// TIA Portal V17 export
// export: Created 2024-09-02T12:50:12.8547271Z, ExportSetting WithDefaults, DisplayName Totally Integrated Automation Portal, DisplayVersion V17, DisplayName TIA Portal Openness, DisplayVersion V17, DisplayName TIA Portal Version Control Interface, DisplayVersion V17, DisplayName STEP 7 Professional, DisplayVersion V17, DisplayName STEP 7 Safety, DisplayVersion V17, DisplayName WinCC Professional, DisplayVersion V17
FUNCTION_BLOCK "AnwFB_Prozess_FG02_BEA3_OP70"   // FB503, LAD
TITLE = Processing dates 2 / Bearbeitungsdaten 2
{ S7_Optimized_Access := 'TRUE' }
AUTHOR : VAF
FAMILY : PROZESS
NAME : PROZESS
VERSION : 0.1
// stored: AutoNumber false, IsIECCheckEnabled false, IsRetainMemResEnabled false, MemoryReserve 100, SetENOAutomatically false, UDAEnableTagReadback false
   VAR
      Station { S7_SetPoint := 'True'} : "SysFB_ProzessDatenStation";
      Gruppe_0 { S7_SetPoint := 'True'} : "SysFB_ProzessDatenGruppe";
      Gruppe_1 { S7_SetPoint := 'True'} : "SysFB_ProzessDatenGruppe";
      Gruppe_2 { S7_SetPoint := 'True'} : "SysFB_ProzessDatenGruppe";
      Gruppe_3 { S7_SetPoint := 'True'} : "SysFB_ProzessDatenGruppe";
   END_VAR
   VAR_TEMP
      t_VKE0 : Bool;
      t_VKE1 : Bool;
      t_Reset : Bool;
      t_Release_Hand_OK : Bool;
      t_Release_Deselect : Bool;
      t_Release_Select : Bool;
      t_Release_NOK_Retry : Bool;
      t_Release_NOK_Reject : Bool;
      t_Reset_Hand_OK : Bool;
      t_Reset_Deselect : Bool;
      t_RetVal_SFC : Int;
   END_VAR
BEGIN

REGION Network 1 (SCL): Reload TAF No/indetyficator / TAF-Nr/Bezeichner umladen
   "AnwDB_ProcessData_FG02_OP70".PROZESS[3].Process.PROC_NR := 3;

   "AnwDB_ProcessData_FG02_OP70".PROZESS[3].Process.DES[1] := 'T';
   "AnwDB_ProcessData_FG02_OP70".PROZESS[3].Process.DES[2] := 'i';
   "AnwDB_ProcessData_FG02_OP70".PROZESS[3].Process.DES[3] := 'g';
   "AnwDB_ProcessData_FG02_OP70".PROZESS[3].Process.DES[4] := 'h';
   "AnwDB_ProcessData_FG02_OP70".PROZESS[3].Process.DES[5] := 't';
   "AnwDB_ProcessData_FG02_OP70".PROZESS[3].Process.DES[6] := 'e';
   "AnwDB_ProcessData_FG02_OP70".PROZESS[3].Process.DES[7] := 'n';
   "AnwDB_ProcessData_FG02_OP70".PROZESS[3].Process.DES[8] := 'i';
   "AnwDB_ProcessData_FG02_OP70".PROZESS[3].Process.DES[9] := 'n';
   "AnwDB_ProcessData_FG02_OP70".PROZESS[3].Process.DES[10] := 'g';
   "AnwDB_ProcessData_FG02_OP70".PROZESS[3].Process.DES[11] := ' ';
   "AnwDB_ProcessData_FG02_OP70".PROZESS[3].Process.DES[12] := ' ';
   "AnwDB_ProcessData_FG02_OP70".PROZESS[3].Process.DES[13] := ' ';
   "AnwDB_ProcessData_FG02_OP70".PROZESS[3].Process.DES[14] := ' ';
   "AnwDB_ProcessData_FG02_OP70".PROZESS[3].Process.DES[15] := ' ';
   "AnwDB_ProcessData_FG02_OP70".PROZESS[3].Process.DES[16] := ' ';
   "AnwDB_ProcessData_FG02_OP70".PROZESS[3].Process.DES[17] := ' ';
   "AnwDB_ProcessData_FG02_OP70".PROZESS[3].Process.DES[18] := ' ';
   "AnwDB_ProcessData_FG02_OP70".PROZESS[3].Process.DES[19] := ' ';
   "AnwDB_ProcessData_FG02_OP70".PROZESS[3].Process.DES[20] := ' ';
   "AnwDB_ProcessData_FG02_OP70".PROZESS[3].Process.DES[21] := ' ';
   "AnwDB_ProcessData_FG02_OP70".PROZESS[3].Process.DES[22] := ' ';
END_REGION

REGION Network 2: VKE0/1
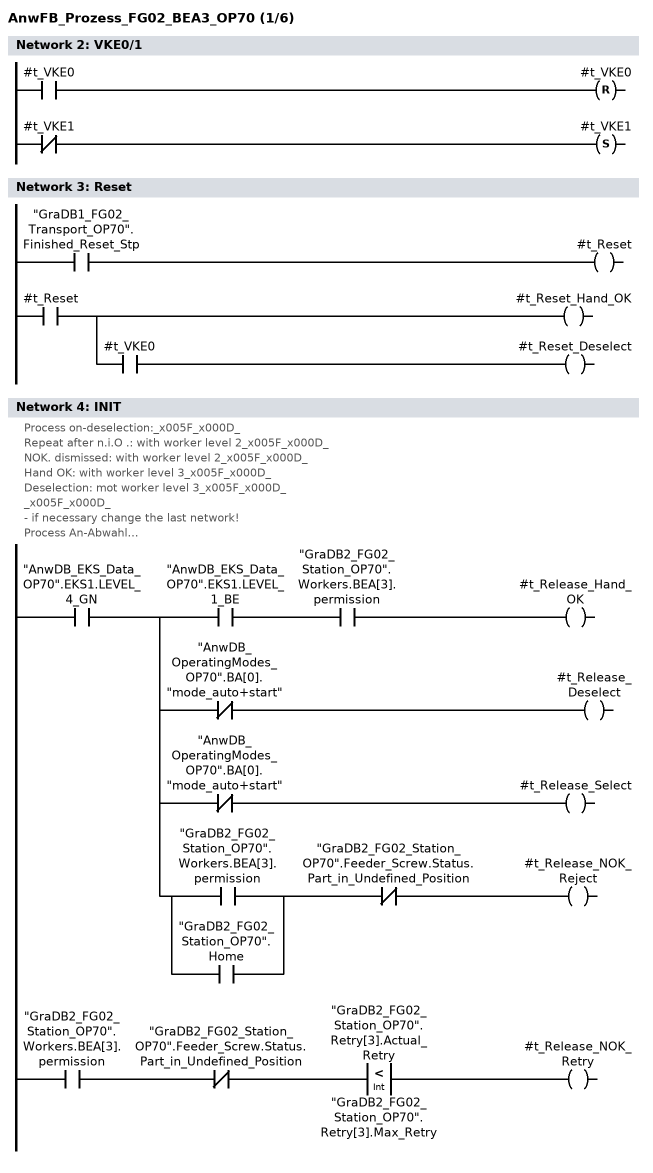
   RUNG wire#powerrail
      Contact( #t_VKE0 )
      R_Coil( #t_VKE0 )
   END_RUNG
   RUNG wire#powerrail
      I_Contact( #t_VKE1 )
      S_Coil( #t_VKE1 )
   END_RUNG
   // the same network as SCL:
   IF #t_VKE0 THEN #t_VKE0 := FALSE; END_IF;
   IF NOT #t_VKE1 THEN #t_VKE1 := TRUE; END_IF;
END_REGION

REGION Network 3: Reset
   RUNG wire#powerrail
      Contact( "GraDB1_FG02_Transport_OP70".Finished_Reset_Stp )
      Coil( #t_Reset )
   END_RUNG
   RUNG wire#powerrail
      Contact( #t_Reset )
      wire#w1
      Coil( #t_Reset_Hand_OK )
   END_RUNG
   RUNG wire#w1
      Contact( #t_VKE0 )
      Coil( #t_Reset_Deselect )
   END_RUNG
   // the same network as SCL:
   #t_Reset := "GraDB1_FG02_Transport_OP70".Finished_Reset_Stp;
   #t_Reset_Hand_OK := #t_Reset;
   #t_Reset_Deselect := #t_Reset AND #t_VKE0;
END_REGION

REGION Network 4: INIT
   // Process on-deselection:_x005F_x000D_
   // Repeat after n.i.O .: with worker level 2_x005F_x000D_
   // NOK. dismissed: with worker level 2_x005F_x000D_
   // Hand OK: with worker level 3_x005F_x000D_
   // Deselection: mot worker level 3_x005F_x000D_
   // _x005F_x000D_
   // - if necessary change the last network!
   // Process An-Abwahl:
   // Wiederholen nach n.i.O.: mit Werkerlevel 2
   // N.i.O. entlassen: mit Werkerlevel 2
   // Hand i.O: mit Werkerlevel 3
   // Abwahl: mot Werkerlevel 3
   // 
   // - bei Änderungen evtl.letztes Netzwerk anpassen !!
   RUNG wire#powerrail
      Contact( "AnwDB_EKS_Data_OP70".EKS1.LEVEL_4_GN )
      wire#w1
      Contact( "AnwDB_EKS_Data_OP70".EKS1.LEVEL_1_BE )
      Contact( "GraDB2_FG02_Station_OP70".Workers.BEA[3].permission )
      Coil( #t_Release_Hand_OK )
   END_RUNG
   RUNG wire#w1
      I_Contact( "AnwDB_OperatingModes_OP70".BA[0]."mode_auto+start" )
      Coil( #t_Release_Deselect )
   END_RUNG
   RUNG wire#w1
      I_Contact( "AnwDB_OperatingModes_OP70".BA[0]."mode_auto+start" )
      Coil( #t_Release_Select )
   END_RUNG
   RUNG wire#w1
      Contact( "GraDB2_FG02_Station_OP70".Workers.BEA[3].permission )
      wire#w2
      I_Contact( "GraDB2_FG02_Station_OP70".Feeder_Screw.Status.Part_in_Undefined_Position )
      Coil( #t_Release_NOK_Reject )
   END_RUNG
   RUNG wire#w1
      Contact( "GraDB2_FG02_Station_OP70".Home )
   END_RUNG wire#w2
   RUNG wire#powerrail
      Contact( "GraDB2_FG02_Station_OP70".Workers.BEA[3].permission )
      I_Contact( "GraDB2_FG02_Station_OP70".Feeder_Screw.Status.Part_in_Undefined_Position )
      { S7_Templates := "SrcType := Int" } LT_Contact(in1 := "GraDB2_FG02_Station_OP70".Retry[3].Actual_Retry, in2 := "GraDB2_FG02_Station_OP70".Retry[3].Max_Retry)
      Coil( #t_Release_NOK_Retry )
   END_RUNG
   // the same network as SCL:
   #t_Release_Hand_OK := "AnwDB_EKS_Data_OP70".EKS1.LEVEL_4_GN AND "AnwDB_EKS_Data_OP70".EKS1.LEVEL_1_BE AND "GraDB2_FG02_Station_OP70".Workers.BEA[3].permission;
   #t_Release_Deselect := "AnwDB_EKS_Data_OP70".EKS1.LEVEL_4_GN AND NOT "AnwDB_OperatingModes_OP70".BA[0]."mode_auto+start";
   #t_Release_Select := "AnwDB_EKS_Data_OP70".EKS1.LEVEL_4_GN AND NOT "AnwDB_OperatingModes_OP70".BA[0]."mode_auto+start";
   #t_Release_NOK_Reject := "AnwDB_EKS_Data_OP70".EKS1.LEVEL_4_GN AND ("GraDB2_FG02_Station_OP70".Workers.BEA[3].permission OR "GraDB2_FG02_Station_OP70".Home) AND NOT "GraDB2_FG02_Station_OP70".Feeder_Screw.Status.Part_in_Undefined_Position;
   #t_Release_NOK_Retry := "GraDB2_FG02_Station_OP70".Workers.BEA[3].permission AND NOT "GraDB2_FG02_Station_OP70".Feeder_Screw.Status.Part_in_Undefined_Position AND ("GraDB2_FG02_Station_OP70".Retry[3].Actual_Retry < "GraDB2_FG02_Station_OP70".Retry[3].Max_Retry);
END_REGION

REGION Network 5: Data Group 0 / Daten Gruppe 0
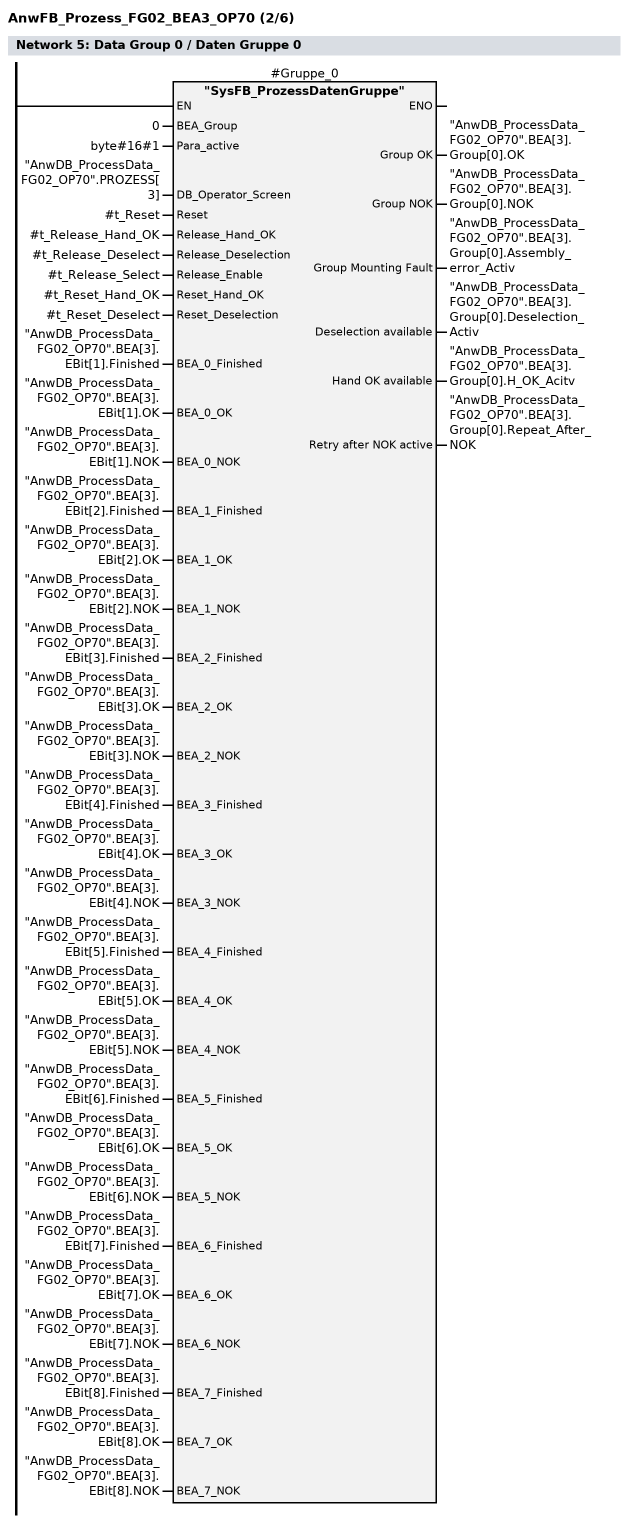
   RUNG wire#powerrail
      #Gruppe_0(BEA_Group := 0, Para_active := byte#16#1, DB_Operator_Screen := "AnwDB_ProcessData_FG02_OP70".PROZESS[3], Reset := #t_Reset, Release_Hand_OK := #t_Release_Hand_OK, Release_Deselection := #t_Release_Deselect, Release_Enable := #t_Release_Select, Reset_Hand_OK := #t_Reset_Hand_OK, Reset_Deselection := #t_Reset_Deselect, BEA_0_Finished := "AnwDB_ProcessData_FG02_OP70".BEA[3].EBit[1].Finished, BEA_0_OK := "AnwDB_ProcessData_FG02_OP70".BEA[3].EBit[1].OK, BEA_0_NOK := "AnwDB_ProcessData_FG02_OP70".BEA[3].EBit[1].NOK, BEA_1_Finished := "AnwDB_ProcessData_FG02_OP70".BEA[3].EBit[2].Finished, BEA_1_OK := "AnwDB_ProcessData_FG02_OP70".BEA[3].EBit[2].OK, BEA_1_NOK := "AnwDB_ProcessData_FG02_OP70".BEA[3].EBit[2].NOK, BEA_2_Finished := "AnwDB_ProcessData_FG02_OP70".BEA[3].EBit[3].Finished, BEA_2_OK := "AnwDB_ProcessData_FG02_OP70".BEA[3].EBit[3].OK, BEA_2_NOK := "AnwDB_ProcessData_FG02_OP70".BEA[3].EBit[3].NOK, BEA_3_Finished := "AnwDB_ProcessData_FG02_OP70".BEA[3].EBit[4].Finished, BEA_3_OK := "AnwDB_ProcessData_FG02_OP70".BEA[3].EBit[4].OK, BEA_3_NOK := "AnwDB_ProcessData_FG02_OP70".BEA[3].EBit[4].NOK, BEA_4_Finished := "AnwDB_ProcessData_FG02_OP70".BEA[3].EBit[5].Finished, BEA_4_OK := "AnwDB_ProcessData_FG02_OP70".BEA[3].EBit[5].OK, BEA_4_NOK := "AnwDB_ProcessData_FG02_OP70".BEA[3].EBit[5].NOK, BEA_5_Finished := "AnwDB_ProcessData_FG02_OP70".BEA[3].EBit[6].Finished, BEA_5_OK := "AnwDB_ProcessData_FG02_OP70".BEA[3].EBit[6].OK, BEA_5_NOK := "AnwDB_ProcessData_FG02_OP70".BEA[3].EBit[6].NOK, BEA_6_Finished := "AnwDB_ProcessData_FG02_OP70".BEA[3].EBit[7].Finished, BEA_6_OK := "AnwDB_ProcessData_FG02_OP70".BEA[3].EBit[7].OK, BEA_6_NOK := "AnwDB_ProcessData_FG02_OP70".BEA[3].EBit[7].NOK, BEA_7_Finished := "AnwDB_ProcessData_FG02_OP70".BEA[3].EBit[8].Finished, BEA_7_OK := "AnwDB_ProcessData_FG02_OP70".BEA[3].EBit[8].OK, BEA_7_NOK := "AnwDB_ProcessData_FG02_OP70".BEA[3].EBit[8].NOK, "Group OK" => "AnwDB_ProcessData_FG02_OP70".BEA[3].Group[0].OK, "Group NOK" => "AnwDB_ProcessData_FG02_OP70".BEA[3].Group[0].NOK, "Group Mounting Fault" => "AnwDB_ProcessData_FG02_OP70".BEA[3].Group[0].Assembly_error_Activ, "Deselection available" => "AnwDB_ProcessData_FG02_OP70".BEA[3].Group[0].Deselection_Activ, "Hand OK available" => "AnwDB_ProcessData_FG02_OP70".BEA[3].Group[0].H_OK_Acitv, "Retry after NOK active" => "AnwDB_ProcessData_FG02_OP70".BEA[3].Group[0].Repeat_After_NOK)
   END_RUNG
   // the same network as SCL:
   #Gruppe_0(BEA_Group := 0,   // "SysFB_ProzessDatenGruppe"
             Para_active := byte#16#1,
             DB_Operator_Screen := "AnwDB_ProcessData_FG02_OP70".PROZESS[3],
             Reset := #t_Reset,
             Release_Hand_OK := #t_Release_Hand_OK,
             Release_Deselection := #t_Release_Deselect,
             Release_Enable := #t_Release_Select,
             Reset_Hand_OK := #t_Reset_Hand_OK,
             Reset_Deselection := #t_Reset_Deselect,
             BEA_0_Finished := "AnwDB_ProcessData_FG02_OP70".BEA[3].EBit[1].Finished,
             BEA_0_OK := "AnwDB_ProcessData_FG02_OP70".BEA[3].EBit[1].OK,
             BEA_0_NOK := "AnwDB_ProcessData_FG02_OP70".BEA[3].EBit[1].NOK,
             BEA_1_Finished := "AnwDB_ProcessData_FG02_OP70".BEA[3].EBit[2].Finished,
             BEA_1_OK := "AnwDB_ProcessData_FG02_OP70".BEA[3].EBit[2].OK,
             BEA_1_NOK := "AnwDB_ProcessData_FG02_OP70".BEA[3].EBit[2].NOK,
             BEA_2_Finished := "AnwDB_ProcessData_FG02_OP70".BEA[3].EBit[3].Finished,
             BEA_2_OK := "AnwDB_ProcessData_FG02_OP70".BEA[3].EBit[3].OK,
             BEA_2_NOK := "AnwDB_ProcessData_FG02_OP70".BEA[3].EBit[3].NOK,
             BEA_3_Finished := "AnwDB_ProcessData_FG02_OP70".BEA[3].EBit[4].Finished,
             BEA_3_OK := "AnwDB_ProcessData_FG02_OP70".BEA[3].EBit[4].OK,
             BEA_3_NOK := "AnwDB_ProcessData_FG02_OP70".BEA[3].EBit[4].NOK,
             BEA_4_Finished := "AnwDB_ProcessData_FG02_OP70".BEA[3].EBit[5].Finished,
             BEA_4_OK := "AnwDB_ProcessData_FG02_OP70".BEA[3].EBit[5].OK,
             BEA_4_NOK := "AnwDB_ProcessData_FG02_OP70".BEA[3].EBit[5].NOK,
             BEA_5_Finished := "AnwDB_ProcessData_FG02_OP70".BEA[3].EBit[6].Finished,
             BEA_5_OK := "AnwDB_ProcessData_FG02_OP70".BEA[3].EBit[6].OK,
             BEA_5_NOK := "AnwDB_ProcessData_FG02_OP70".BEA[3].EBit[6].NOK,
             BEA_6_Finished := "AnwDB_ProcessData_FG02_OP70".BEA[3].EBit[7].Finished,
             BEA_6_OK := "AnwDB_ProcessData_FG02_OP70".BEA[3].EBit[7].OK,
             BEA_6_NOK := "AnwDB_ProcessData_FG02_OP70".BEA[3].EBit[7].NOK,
             BEA_7_Finished := "AnwDB_ProcessData_FG02_OP70".BEA[3].EBit[8].Finished,
             BEA_7_OK := "AnwDB_ProcessData_FG02_OP70".BEA[3].EBit[8].OK,
             BEA_7_NOK := "AnwDB_ProcessData_FG02_OP70".BEA[3].EBit[8].NOK,
             "Group OK" => "AnwDB_ProcessData_FG02_OP70".BEA[3].Group[0].OK,
             "Group NOK" => "AnwDB_ProcessData_FG02_OP70".BEA[3].Group[0].NOK,
             "Group Mounting Fault" => "AnwDB_ProcessData_FG02_OP70".BEA[3].Group[0].Assembly_error_Activ,
             "Deselection available" => "AnwDB_ProcessData_FG02_OP70".BEA[3].Group[0].Deselection_Activ,
             "Hand OK available" => "AnwDB_ProcessData_FG02_OP70".BEA[3].Group[0].H_OK_Acitv,
             "Retry after NOK active" => "AnwDB_ProcessData_FG02_OP70".BEA[3].Group[0].Repeat_After_NOK);
END_REGION

REGION Network 6: Data Group 1 / Daten Gruppe 1
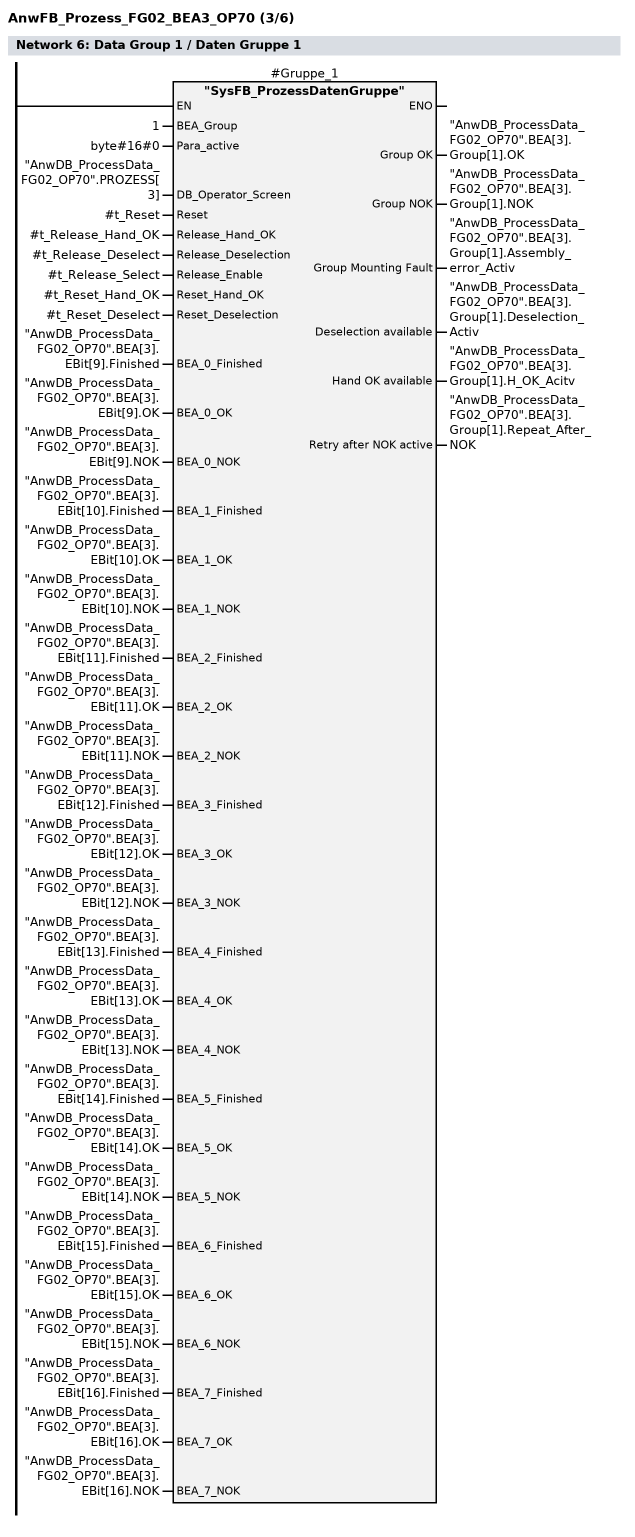
   RUNG wire#powerrail
      #Gruppe_1(BEA_Group := 1, Para_active := byte#16#0, DB_Operator_Screen := "AnwDB_ProcessData_FG02_OP70".PROZESS[3], Reset := #t_Reset, Release_Hand_OK := #t_Release_Hand_OK, Release_Deselection := #t_Release_Deselect, Release_Enable := #t_Release_Select, Reset_Hand_OK := #t_Reset_Hand_OK, Reset_Deselection := #t_Reset_Deselect, BEA_0_Finished := "AnwDB_ProcessData_FG02_OP70".BEA[3].EBit[9].Finished, BEA_0_OK := "AnwDB_ProcessData_FG02_OP70".BEA[3].EBit[9].OK, BEA_0_NOK := "AnwDB_ProcessData_FG02_OP70".BEA[3].EBit[9].NOK, BEA_1_Finished := "AnwDB_ProcessData_FG02_OP70".BEA[3].EBit[10].Finished, BEA_1_OK := "AnwDB_ProcessData_FG02_OP70".BEA[3].EBit[10].OK, BEA_1_NOK := "AnwDB_ProcessData_FG02_OP70".BEA[3].EBit[10].NOK, BEA_2_Finished := "AnwDB_ProcessData_FG02_OP70".BEA[3].EBit[11].Finished, BEA_2_OK := "AnwDB_ProcessData_FG02_OP70".BEA[3].EBit[11].OK, BEA_2_NOK := "AnwDB_ProcessData_FG02_OP70".BEA[3].EBit[11].NOK, BEA_3_Finished := "AnwDB_ProcessData_FG02_OP70".BEA[3].EBit[12].Finished, BEA_3_OK := "AnwDB_ProcessData_FG02_OP70".BEA[3].EBit[12].OK, BEA_3_NOK := "AnwDB_ProcessData_FG02_OP70".BEA[3].EBit[12].NOK, BEA_4_Finished := "AnwDB_ProcessData_FG02_OP70".BEA[3].EBit[13].Finished, BEA_4_OK := "AnwDB_ProcessData_FG02_OP70".BEA[3].EBit[13].OK, BEA_4_NOK := "AnwDB_ProcessData_FG02_OP70".BEA[3].EBit[13].NOK, BEA_5_Finished := "AnwDB_ProcessData_FG02_OP70".BEA[3].EBit[14].Finished, BEA_5_OK := "AnwDB_ProcessData_FG02_OP70".BEA[3].EBit[14].OK, BEA_5_NOK := "AnwDB_ProcessData_FG02_OP70".BEA[3].EBit[14].NOK, BEA_6_Finished := "AnwDB_ProcessData_FG02_OP70".BEA[3].EBit[15].Finished, BEA_6_OK := "AnwDB_ProcessData_FG02_OP70".BEA[3].EBit[15].OK, BEA_6_NOK := "AnwDB_ProcessData_FG02_OP70".BEA[3].EBit[15].NOK, BEA_7_Finished := "AnwDB_ProcessData_FG02_OP70".BEA[3].EBit[16].Finished, BEA_7_OK := "AnwDB_ProcessData_FG02_OP70".BEA[3].EBit[16].OK, BEA_7_NOK := "AnwDB_ProcessData_FG02_OP70".BEA[3].EBit[16].NOK, "Group OK" => "AnwDB_ProcessData_FG02_OP70".BEA[3].Group[1].OK, "Group NOK" => "AnwDB_ProcessData_FG02_OP70".BEA[3].Group[1].NOK, "Group Mounting Fault" => "AnwDB_ProcessData_FG02_OP70".BEA[3].Group[1].Assembly_error_Activ, "Deselection available" => "AnwDB_ProcessData_FG02_OP70".BEA[3].Group[1].Deselection_Activ, "Hand OK available" => "AnwDB_ProcessData_FG02_OP70".BEA[3].Group[1].H_OK_Acitv, "Retry after NOK active" => "AnwDB_ProcessData_FG02_OP70".BEA[3].Group[1].Repeat_After_NOK)
   END_RUNG
   // the same network as SCL:
   #Gruppe_1(BEA_Group := 1,   // "SysFB_ProzessDatenGruppe"
             Para_active := byte#16#0,
             DB_Operator_Screen := "AnwDB_ProcessData_FG02_OP70".PROZESS[3],
             Reset := #t_Reset,
             Release_Hand_OK := #t_Release_Hand_OK,
             Release_Deselection := #t_Release_Deselect,
             Release_Enable := #t_Release_Select,
             Reset_Hand_OK := #t_Reset_Hand_OK,
             Reset_Deselection := #t_Reset_Deselect,
             BEA_0_Finished := "AnwDB_ProcessData_FG02_OP70".BEA[3].EBit[9].Finished,
             BEA_0_OK := "AnwDB_ProcessData_FG02_OP70".BEA[3].EBit[9].OK,
             BEA_0_NOK := "AnwDB_ProcessData_FG02_OP70".BEA[3].EBit[9].NOK,
             BEA_1_Finished := "AnwDB_ProcessData_FG02_OP70".BEA[3].EBit[10].Finished,
             BEA_1_OK := "AnwDB_ProcessData_FG02_OP70".BEA[3].EBit[10].OK,
             BEA_1_NOK := "AnwDB_ProcessData_FG02_OP70".BEA[3].EBit[10].NOK,
             BEA_2_Finished := "AnwDB_ProcessData_FG02_OP70".BEA[3].EBit[11].Finished,
             BEA_2_OK := "AnwDB_ProcessData_FG02_OP70".BEA[3].EBit[11].OK,
             BEA_2_NOK := "AnwDB_ProcessData_FG02_OP70".BEA[3].EBit[11].NOK,
             BEA_3_Finished := "AnwDB_ProcessData_FG02_OP70".BEA[3].EBit[12].Finished,
             BEA_3_OK := "AnwDB_ProcessData_FG02_OP70".BEA[3].EBit[12].OK,
             BEA_3_NOK := "AnwDB_ProcessData_FG02_OP70".BEA[3].EBit[12].NOK,
             BEA_4_Finished := "AnwDB_ProcessData_FG02_OP70".BEA[3].EBit[13].Finished,
             BEA_4_OK := "AnwDB_ProcessData_FG02_OP70".BEA[3].EBit[13].OK,
             BEA_4_NOK := "AnwDB_ProcessData_FG02_OP70".BEA[3].EBit[13].NOK,
             BEA_5_Finished := "AnwDB_ProcessData_FG02_OP70".BEA[3].EBit[14].Finished,
             BEA_5_OK := "AnwDB_ProcessData_FG02_OP70".BEA[3].EBit[14].OK,
             BEA_5_NOK := "AnwDB_ProcessData_FG02_OP70".BEA[3].EBit[14].NOK,
             BEA_6_Finished := "AnwDB_ProcessData_FG02_OP70".BEA[3].EBit[15].Finished,
             BEA_6_OK := "AnwDB_ProcessData_FG02_OP70".BEA[3].EBit[15].OK,
             BEA_6_NOK := "AnwDB_ProcessData_FG02_OP70".BEA[3].EBit[15].NOK,
             BEA_7_Finished := "AnwDB_ProcessData_FG02_OP70".BEA[3].EBit[16].Finished,
             BEA_7_OK := "AnwDB_ProcessData_FG02_OP70".BEA[3].EBit[16].OK,
             BEA_7_NOK := "AnwDB_ProcessData_FG02_OP70".BEA[3].EBit[16].NOK,
             "Group OK" => "AnwDB_ProcessData_FG02_OP70".BEA[3].Group[1].OK,
             "Group NOK" => "AnwDB_ProcessData_FG02_OP70".BEA[3].Group[1].NOK,
             "Group Mounting Fault" => "AnwDB_ProcessData_FG02_OP70".BEA[3].Group[1].Assembly_error_Activ,
             "Deselection available" => "AnwDB_ProcessData_FG02_OP70".BEA[3].Group[1].Deselection_Activ,
             "Hand OK available" => "AnwDB_ProcessData_FG02_OP70".BEA[3].Group[1].H_OK_Acitv,
             "Retry after NOK active" => "AnwDB_ProcessData_FG02_OP70".BEA[3].Group[1].Repeat_After_NOK);
END_REGION

REGION Network 7: Data Group 2 / Daten Gruppe 2
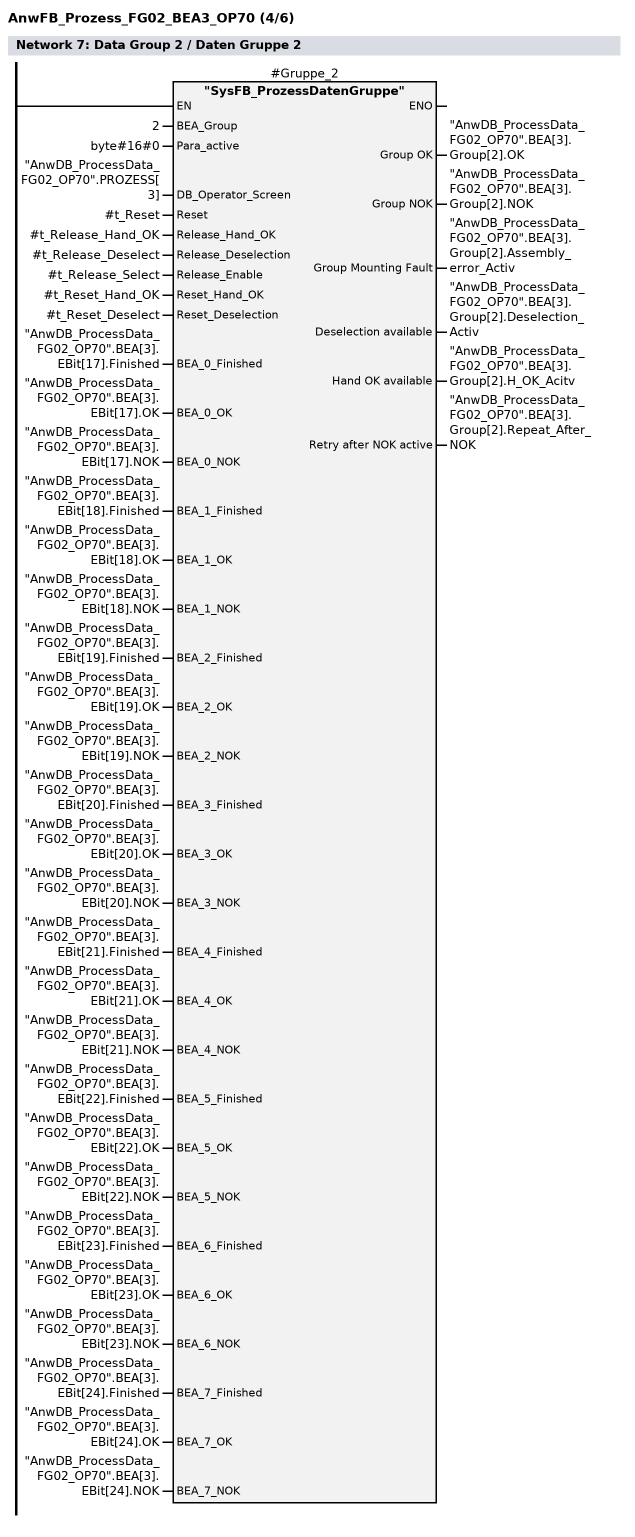
   RUNG wire#powerrail
      #Gruppe_2(BEA_Group := 2, Para_active := byte#16#0, DB_Operator_Screen := "AnwDB_ProcessData_FG02_OP70".PROZESS[3], Reset := #t_Reset, Release_Hand_OK := #t_Release_Hand_OK, Release_Deselection := #t_Release_Deselect, Release_Enable := #t_Release_Select, Reset_Hand_OK := #t_Reset_Hand_OK, Reset_Deselection := #t_Reset_Deselect, BEA_0_Finished := "AnwDB_ProcessData_FG02_OP70".BEA[3].EBit[17].Finished, BEA_0_OK := "AnwDB_ProcessData_FG02_OP70".BEA[3].EBit[17].OK, BEA_0_NOK := "AnwDB_ProcessData_FG02_OP70".BEA[3].EBit[17].NOK, BEA_1_Finished := "AnwDB_ProcessData_FG02_OP70".BEA[3].EBit[18].Finished, BEA_1_OK := "AnwDB_ProcessData_FG02_OP70".BEA[3].EBit[18].OK, BEA_1_NOK := "AnwDB_ProcessData_FG02_OP70".BEA[3].EBit[18].NOK, BEA_2_Finished := "AnwDB_ProcessData_FG02_OP70".BEA[3].EBit[19].Finished, BEA_2_OK := "AnwDB_ProcessData_FG02_OP70".BEA[3].EBit[19].OK, BEA_2_NOK := "AnwDB_ProcessData_FG02_OP70".BEA[3].EBit[19].NOK, BEA_3_Finished := "AnwDB_ProcessData_FG02_OP70".BEA[3].EBit[20].Finished, BEA_3_OK := "AnwDB_ProcessData_FG02_OP70".BEA[3].EBit[20].OK, BEA_3_NOK := "AnwDB_ProcessData_FG02_OP70".BEA[3].EBit[20].NOK, BEA_4_Finished := "AnwDB_ProcessData_FG02_OP70".BEA[3].EBit[21].Finished, BEA_4_OK := "AnwDB_ProcessData_FG02_OP70".BEA[3].EBit[21].OK, BEA_4_NOK := "AnwDB_ProcessData_FG02_OP70".BEA[3].EBit[21].NOK, BEA_5_Finished := "AnwDB_ProcessData_FG02_OP70".BEA[3].EBit[22].Finished, BEA_5_OK := "AnwDB_ProcessData_FG02_OP70".BEA[3].EBit[22].OK, BEA_5_NOK := "AnwDB_ProcessData_FG02_OP70".BEA[3].EBit[22].NOK, BEA_6_Finished := "AnwDB_ProcessData_FG02_OP70".BEA[3].EBit[23].Finished, BEA_6_OK := "AnwDB_ProcessData_FG02_OP70".BEA[3].EBit[23].OK, BEA_6_NOK := "AnwDB_ProcessData_FG02_OP70".BEA[3].EBit[23].NOK, BEA_7_Finished := "AnwDB_ProcessData_FG02_OP70".BEA[3].EBit[24].Finished, BEA_7_OK := "AnwDB_ProcessData_FG02_OP70".BEA[3].EBit[24].OK, BEA_7_NOK := "AnwDB_ProcessData_FG02_OP70".BEA[3].EBit[24].NOK, "Group OK" => "AnwDB_ProcessData_FG02_OP70".BEA[3].Group[2].OK, "Group NOK" => "AnwDB_ProcessData_FG02_OP70".BEA[3].Group[2].NOK, "Group Mounting Fault" => "AnwDB_ProcessData_FG02_OP70".BEA[3].Group[2].Assembly_error_Activ, "Deselection available" => "AnwDB_ProcessData_FG02_OP70".BEA[3].Group[2].Deselection_Activ, "Hand OK available" => "AnwDB_ProcessData_FG02_OP70".BEA[3].Group[2].H_OK_Acitv, "Retry after NOK active" => "AnwDB_ProcessData_FG02_OP70".BEA[3].Group[2].Repeat_After_NOK)
   END_RUNG
   // the same network as SCL:
   #Gruppe_2(BEA_Group := 2,   // "SysFB_ProzessDatenGruppe"
             Para_active := byte#16#0,
             DB_Operator_Screen := "AnwDB_ProcessData_FG02_OP70".PROZESS[3],
             Reset := #t_Reset,
             Release_Hand_OK := #t_Release_Hand_OK,
             Release_Deselection := #t_Release_Deselect,
             Release_Enable := #t_Release_Select,
             Reset_Hand_OK := #t_Reset_Hand_OK,
             Reset_Deselection := #t_Reset_Deselect,
             BEA_0_Finished := "AnwDB_ProcessData_FG02_OP70".BEA[3].EBit[17].Finished,
             BEA_0_OK := "AnwDB_ProcessData_FG02_OP70".BEA[3].EBit[17].OK,
             BEA_0_NOK := "AnwDB_ProcessData_FG02_OP70".BEA[3].EBit[17].NOK,
             BEA_1_Finished := "AnwDB_ProcessData_FG02_OP70".BEA[3].EBit[18].Finished,
             BEA_1_OK := "AnwDB_ProcessData_FG02_OP70".BEA[3].EBit[18].OK,
             BEA_1_NOK := "AnwDB_ProcessData_FG02_OP70".BEA[3].EBit[18].NOK,
             BEA_2_Finished := "AnwDB_ProcessData_FG02_OP70".BEA[3].EBit[19].Finished,
             BEA_2_OK := "AnwDB_ProcessData_FG02_OP70".BEA[3].EBit[19].OK,
             BEA_2_NOK := "AnwDB_ProcessData_FG02_OP70".BEA[3].EBit[19].NOK,
             BEA_3_Finished := "AnwDB_ProcessData_FG02_OP70".BEA[3].EBit[20].Finished,
             BEA_3_OK := "AnwDB_ProcessData_FG02_OP70".BEA[3].EBit[20].OK,
             BEA_3_NOK := "AnwDB_ProcessData_FG02_OP70".BEA[3].EBit[20].NOK,
             BEA_4_Finished := "AnwDB_ProcessData_FG02_OP70".BEA[3].EBit[21].Finished,
             BEA_4_OK := "AnwDB_ProcessData_FG02_OP70".BEA[3].EBit[21].OK,
             BEA_4_NOK := "AnwDB_ProcessData_FG02_OP70".BEA[3].EBit[21].NOK,
             BEA_5_Finished := "AnwDB_ProcessData_FG02_OP70".BEA[3].EBit[22].Finished,
             BEA_5_OK := "AnwDB_ProcessData_FG02_OP70".BEA[3].EBit[22].OK,
             BEA_5_NOK := "AnwDB_ProcessData_FG02_OP70".BEA[3].EBit[22].NOK,
             BEA_6_Finished := "AnwDB_ProcessData_FG02_OP70".BEA[3].EBit[23].Finished,
             BEA_6_OK := "AnwDB_ProcessData_FG02_OP70".BEA[3].EBit[23].OK,
             BEA_6_NOK := "AnwDB_ProcessData_FG02_OP70".BEA[3].EBit[23].NOK,
             BEA_7_Finished := "AnwDB_ProcessData_FG02_OP70".BEA[3].EBit[24].Finished,
             BEA_7_OK := "AnwDB_ProcessData_FG02_OP70".BEA[3].EBit[24].OK,
             BEA_7_NOK := "AnwDB_ProcessData_FG02_OP70".BEA[3].EBit[24].NOK,
             "Group OK" => "AnwDB_ProcessData_FG02_OP70".BEA[3].Group[2].OK,
             "Group NOK" => "AnwDB_ProcessData_FG02_OP70".BEA[3].Group[2].NOK,
             "Group Mounting Fault" => "AnwDB_ProcessData_FG02_OP70".BEA[3].Group[2].Assembly_error_Activ,
             "Deselection available" => "AnwDB_ProcessData_FG02_OP70".BEA[3].Group[2].Deselection_Activ,
             "Hand OK available" => "AnwDB_ProcessData_FG02_OP70".BEA[3].Group[2].H_OK_Acitv,
             "Retry after NOK active" => "AnwDB_ProcessData_FG02_OP70".BEA[3].Group[2].Repeat_After_NOK);
END_REGION

REGION Network 8: Data Group 3 / Daten Gruppe 3
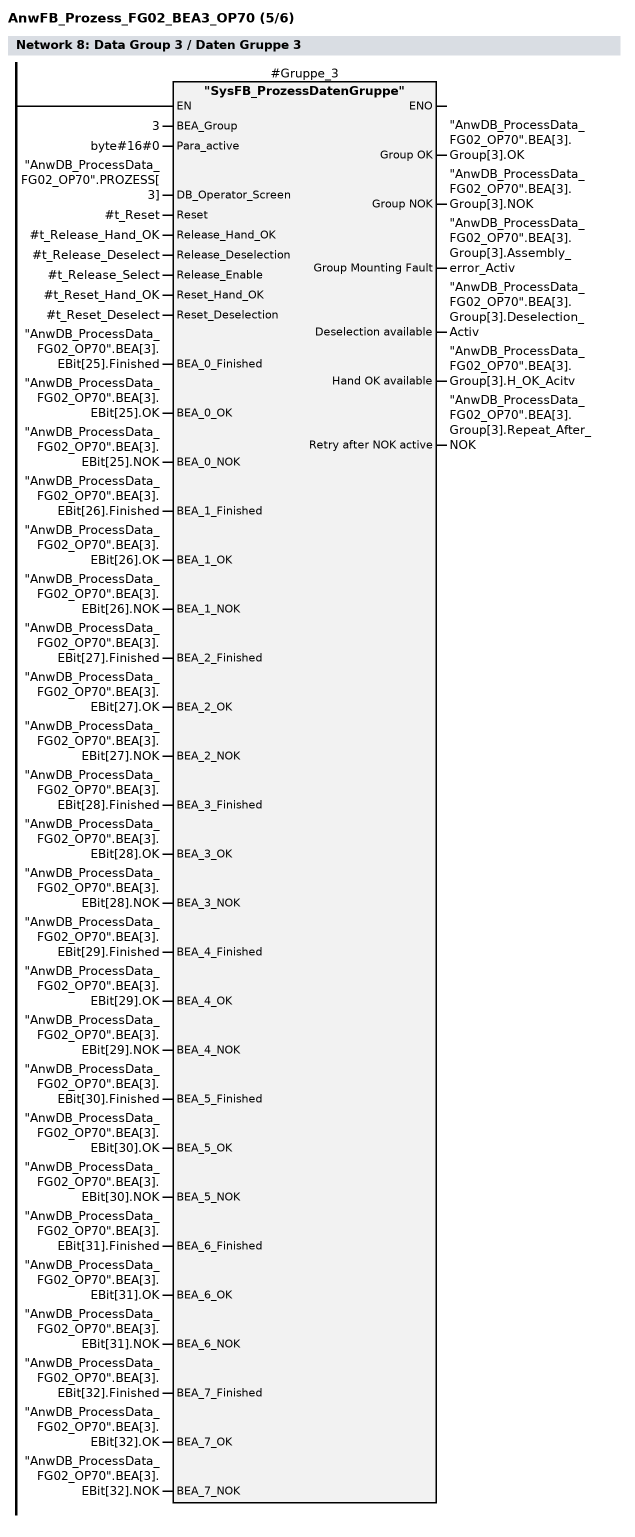
   RUNG wire#powerrail
      #Gruppe_3(BEA_Group := 3, Para_active := byte#16#0, DB_Operator_Screen := "AnwDB_ProcessData_FG02_OP70".PROZESS[3], Reset := #t_Reset, Release_Hand_OK := #t_Release_Hand_OK, Release_Deselection := #t_Release_Deselect, Release_Enable := #t_Release_Select, Reset_Hand_OK := #t_Reset_Hand_OK, Reset_Deselection := #t_Reset_Deselect, BEA_0_Finished := "AnwDB_ProcessData_FG02_OP70".BEA[3].EBit[25].Finished, BEA_0_OK := "AnwDB_ProcessData_FG02_OP70".BEA[3].EBit[25].OK, BEA_0_NOK := "AnwDB_ProcessData_FG02_OP70".BEA[3].EBit[25].NOK, BEA_1_Finished := "AnwDB_ProcessData_FG02_OP70".BEA[3].EBit[26].Finished, BEA_1_OK := "AnwDB_ProcessData_FG02_OP70".BEA[3].EBit[26].OK, BEA_1_NOK := "AnwDB_ProcessData_FG02_OP70".BEA[3].EBit[26].NOK, BEA_2_Finished := "AnwDB_ProcessData_FG02_OP70".BEA[3].EBit[27].Finished, BEA_2_OK := "AnwDB_ProcessData_FG02_OP70".BEA[3].EBit[27].OK, BEA_2_NOK := "AnwDB_ProcessData_FG02_OP70".BEA[3].EBit[27].NOK, BEA_3_Finished := "AnwDB_ProcessData_FG02_OP70".BEA[3].EBit[28].Finished, BEA_3_OK := "AnwDB_ProcessData_FG02_OP70".BEA[3].EBit[28].OK, BEA_3_NOK := "AnwDB_ProcessData_FG02_OP70".BEA[3].EBit[28].NOK, BEA_4_Finished := "AnwDB_ProcessData_FG02_OP70".BEA[3].EBit[29].Finished, BEA_4_OK := "AnwDB_ProcessData_FG02_OP70".BEA[3].EBit[29].OK, BEA_4_NOK := "AnwDB_ProcessData_FG02_OP70".BEA[3].EBit[29].NOK, BEA_5_Finished := "AnwDB_ProcessData_FG02_OP70".BEA[3].EBit[30].Finished, BEA_5_OK := "AnwDB_ProcessData_FG02_OP70".BEA[3].EBit[30].OK, BEA_5_NOK := "AnwDB_ProcessData_FG02_OP70".BEA[3].EBit[30].NOK, BEA_6_Finished := "AnwDB_ProcessData_FG02_OP70".BEA[3].EBit[31].Finished, BEA_6_OK := "AnwDB_ProcessData_FG02_OP70".BEA[3].EBit[31].OK, BEA_6_NOK := "AnwDB_ProcessData_FG02_OP70".BEA[3].EBit[31].NOK, BEA_7_Finished := "AnwDB_ProcessData_FG02_OP70".BEA[3].EBit[32].Finished, BEA_7_OK := "AnwDB_ProcessData_FG02_OP70".BEA[3].EBit[32].OK, BEA_7_NOK := "AnwDB_ProcessData_FG02_OP70".BEA[3].EBit[32].NOK, "Group OK" => "AnwDB_ProcessData_FG02_OP70".BEA[3].Group[3].OK, "Group NOK" => "AnwDB_ProcessData_FG02_OP70".BEA[3].Group[3].NOK, "Group Mounting Fault" => "AnwDB_ProcessData_FG02_OP70".BEA[3].Group[3].Assembly_error_Activ, "Deselection available" => "AnwDB_ProcessData_FG02_OP70".BEA[3].Group[3].Deselection_Activ, "Hand OK available" => "AnwDB_ProcessData_FG02_OP70".BEA[3].Group[3].H_OK_Acitv, "Retry after NOK active" => "AnwDB_ProcessData_FG02_OP70".BEA[3].Group[3].Repeat_After_NOK)
   END_RUNG
   // the same network as SCL:
   #Gruppe_3(BEA_Group := 3,   // "SysFB_ProzessDatenGruppe"
             Para_active := byte#16#0,
             DB_Operator_Screen := "AnwDB_ProcessData_FG02_OP70".PROZESS[3],
             Reset := #t_Reset,
             Release_Hand_OK := #t_Release_Hand_OK,
             Release_Deselection := #t_Release_Deselect,
             Release_Enable := #t_Release_Select,
             Reset_Hand_OK := #t_Reset_Hand_OK,
             Reset_Deselection := #t_Reset_Deselect,
             BEA_0_Finished := "AnwDB_ProcessData_FG02_OP70".BEA[3].EBit[25].Finished,
             BEA_0_OK := "AnwDB_ProcessData_FG02_OP70".BEA[3].EBit[25].OK,
             BEA_0_NOK := "AnwDB_ProcessData_FG02_OP70".BEA[3].EBit[25].NOK,
             BEA_1_Finished := "AnwDB_ProcessData_FG02_OP70".BEA[3].EBit[26].Finished,
             BEA_1_OK := "AnwDB_ProcessData_FG02_OP70".BEA[3].EBit[26].OK,
             BEA_1_NOK := "AnwDB_ProcessData_FG02_OP70".BEA[3].EBit[26].NOK,
             BEA_2_Finished := "AnwDB_ProcessData_FG02_OP70".BEA[3].EBit[27].Finished,
             BEA_2_OK := "AnwDB_ProcessData_FG02_OP70".BEA[3].EBit[27].OK,
             BEA_2_NOK := "AnwDB_ProcessData_FG02_OP70".BEA[3].EBit[27].NOK,
             BEA_3_Finished := "AnwDB_ProcessData_FG02_OP70".BEA[3].EBit[28].Finished,
             BEA_3_OK := "AnwDB_ProcessData_FG02_OP70".BEA[3].EBit[28].OK,
             BEA_3_NOK := "AnwDB_ProcessData_FG02_OP70".BEA[3].EBit[28].NOK,
             BEA_4_Finished := "AnwDB_ProcessData_FG02_OP70".BEA[3].EBit[29].Finished,
             BEA_4_OK := "AnwDB_ProcessData_FG02_OP70".BEA[3].EBit[29].OK,
             BEA_4_NOK := "AnwDB_ProcessData_FG02_OP70".BEA[3].EBit[29].NOK,
             BEA_5_Finished := "AnwDB_ProcessData_FG02_OP70".BEA[3].EBit[30].Finished,
             BEA_5_OK := "AnwDB_ProcessData_FG02_OP70".BEA[3].EBit[30].OK,
             BEA_5_NOK := "AnwDB_ProcessData_FG02_OP70".BEA[3].EBit[30].NOK,
             BEA_6_Finished := "AnwDB_ProcessData_FG02_OP70".BEA[3].EBit[31].Finished,
             BEA_6_OK := "AnwDB_ProcessData_FG02_OP70".BEA[3].EBit[31].OK,
             BEA_6_NOK := "AnwDB_ProcessData_FG02_OP70".BEA[3].EBit[31].NOK,
             BEA_7_Finished := "AnwDB_ProcessData_FG02_OP70".BEA[3].EBit[32].Finished,
             BEA_7_OK := "AnwDB_ProcessData_FG02_OP70".BEA[3].EBit[32].OK,
             BEA_7_NOK := "AnwDB_ProcessData_FG02_OP70".BEA[3].EBit[32].NOK,
             "Group OK" => "AnwDB_ProcessData_FG02_OP70".BEA[3].Group[3].OK,
             "Group NOK" => "AnwDB_ProcessData_FG02_OP70".BEA[3].Group[3].NOK,
             "Group Mounting Fault" => "AnwDB_ProcessData_FG02_OP70".BEA[3].Group[3].Assembly_error_Activ,
             "Deselection available" => "AnwDB_ProcessData_FG02_OP70".BEA[3].Group[3].Deselection_Activ,
             "Hand OK available" => "AnwDB_ProcessData_FG02_OP70".BEA[3].Group[3].H_OK_Acitv,
             "Retry after NOK active" => "AnwDB_ProcessData_FG02_OP70".BEA[3].Group[3].Repeat_After_NOK);
END_REGION

REGION Network 9: Reset Started
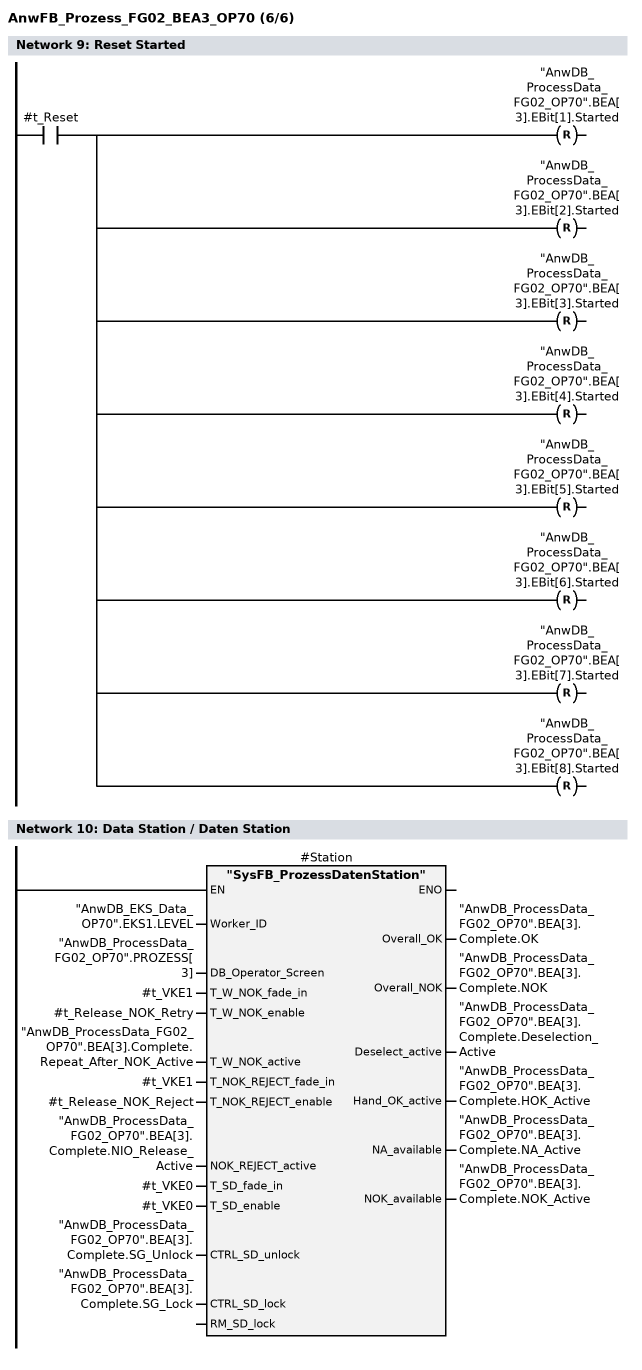
   RUNG wire#powerrail
      Contact( #t_Reset )
      wire#w1
      R_Coil( "AnwDB_ProcessData_FG02_OP70".BEA[3].EBit[1].Started )
   END_RUNG
   RUNG wire#w1
      R_Coil( "AnwDB_ProcessData_FG02_OP70".BEA[3].EBit[2].Started )
   END_RUNG
   RUNG wire#w1
      R_Coil( "AnwDB_ProcessData_FG02_OP70".BEA[3].EBit[3].Started )
   END_RUNG
   RUNG wire#w1
      R_Coil( "AnwDB_ProcessData_FG02_OP70".BEA[3].EBit[4].Started )
   END_RUNG
   RUNG wire#w1
      R_Coil( "AnwDB_ProcessData_FG02_OP70".BEA[3].EBit[5].Started )
   END_RUNG
   RUNG wire#w1
      R_Coil( "AnwDB_ProcessData_FG02_OP70".BEA[3].EBit[6].Started )
   END_RUNG
   RUNG wire#w1
      R_Coil( "AnwDB_ProcessData_FG02_OP70".BEA[3].EBit[7].Started )
   END_RUNG
   RUNG wire#w1
      R_Coil( "AnwDB_ProcessData_FG02_OP70".BEA[3].EBit[8].Started )
   END_RUNG
   // the same network as SCL:
   IF #t_Reset THEN
       "AnwDB_ProcessData_FG02_OP70".BEA[3].EBit[1].Started := FALSE;
       "AnwDB_ProcessData_FG02_OP70".BEA[3].EBit[2].Started := FALSE;
       "AnwDB_ProcessData_FG02_OP70".BEA[3].EBit[3].Started := FALSE;
       "AnwDB_ProcessData_FG02_OP70".BEA[3].EBit[4].Started := FALSE;
       "AnwDB_ProcessData_FG02_OP70".BEA[3].EBit[5].Started := FALSE;
       "AnwDB_ProcessData_FG02_OP70".BEA[3].EBit[6].Started := FALSE;
       "AnwDB_ProcessData_FG02_OP70".BEA[3].EBit[7].Started := FALSE;
       "AnwDB_ProcessData_FG02_OP70".BEA[3].EBit[8].Started := FALSE;
   END_IF;
END_REGION

REGION Network 10: Data Station / Daten Station
   RUNG wire#powerrail
      #Station(Worker_ID := "AnwDB_EKS_Data_OP70".EKS1.LEVEL, DB_Operator_Screen := "AnwDB_ProcessData_FG02_OP70".PROZESS[3], T_W_NOK_fade_in := #t_VKE1, T_W_NOK_enable := #t_Release_NOK_Retry, T_W_NOK_active := "AnwDB_ProcessData_FG02_OP70".BEA[3].Complete.Repeat_After_NOK_Active, T_NOK_REJECT_fade_in := #t_VKE1, T_NOK_REJECT_enable := #t_Release_NOK_Reject, NOK_REJECT_active := "AnwDB_ProcessData_FG02_OP70".BEA[3].Complete.NIO_Release_Active, T_SD_fade_in := #t_VKE0, T_SD_enable := #t_VKE0, CTRL_SD_unlock := "AnwDB_ProcessData_FG02_OP70".BEA[3].Complete.SG_Unlock, CTRL_SD_lock := "AnwDB_ProcessData_FG02_OP70".BEA[3].Complete.SG_Lock, RM_SD_lock :=, Overall_OK => "AnwDB_ProcessData_FG02_OP70".BEA[3].Complete.OK, Overall_NOK => "AnwDB_ProcessData_FG02_OP70".BEA[3].Complete.NOK, Deselect_active => "AnwDB_ProcessData_FG02_OP70".BEA[3].Complete.Deselection_Active, Hand_OK_active => "AnwDB_ProcessData_FG02_OP70".BEA[3].Complete.HOK_Active, NA_available => "AnwDB_ProcessData_FG02_OP70".BEA[3].Complete.NA_Active, NOK_available => "AnwDB_ProcessData_FG02_OP70".BEA[3].Complete.NOK_Active)
   END_RUNG
   // the same network as SCL:
   #Station(Worker_ID := "AnwDB_EKS_Data_OP70".EKS1.LEVEL,   // "SysFB_ProzessDatenStation"
            DB_Operator_Screen := "AnwDB_ProcessData_FG02_OP70".PROZESS[3],
            T_W_NOK_fade_in := #t_VKE1,
            T_W_NOK_enable := #t_Release_NOK_Retry,
            T_W_NOK_active := "AnwDB_ProcessData_FG02_OP70".BEA[3].Complete.Repeat_After_NOK_Active,
            T_NOK_REJECT_fade_in := #t_VKE1,
            T_NOK_REJECT_enable := #t_Release_NOK_Reject,
            NOK_REJECT_active := "AnwDB_ProcessData_FG02_OP70".BEA[3].Complete.NIO_Release_Active,
            T_SD_fade_in := #t_VKE0,
            T_SD_enable := #t_VKE0,
            CTRL_SD_unlock := "AnwDB_ProcessData_FG02_OP70".BEA[3].Complete.SG_Unlock,
            CTRL_SD_lock := "AnwDB_ProcessData_FG02_OP70".BEA[3].Complete.SG_Lock,
            Overall_OK => "AnwDB_ProcessData_FG02_OP70".BEA[3].Complete.OK,
            Overall_NOK => "AnwDB_ProcessData_FG02_OP70".BEA[3].Complete.NOK,
            Deselect_active => "AnwDB_ProcessData_FG02_OP70".BEA[3].Complete.Deselection_Active,
            Hand_OK_active => "AnwDB_ProcessData_FG02_OP70".BEA[3].Complete.HOK_Active,
            NA_available => "AnwDB_ProcessData_FG02_OP70".BEA[3].Complete.NA_Active,
            NOK_available => "AnwDB_ProcessData_FG02_OP70".BEA[3].Complete.NOK_Active);
END_REGION
END_FUNCTION_BLOCK
